// TIA Portal V15.1 export
// export: Created 2020-06-12T07:35:49.5849609Z, ExportSetting None, DisplayName Totally Integrated Automation Portal, DisplayVersion V15.1, DisplayName TIA Portal Openness, DisplayVersion V15.1, DisplayName STEP 7 Professional, DisplayVersion V15.1, DisplayName STEP 7 Safety, DisplayVersion V15.1, DisplayName WinCC Advanced, DisplayVersion V15.1
FUNCTION "MELT_Call" : Void   // FC91, FBD
{ S7_Optimized_Access := 'TRUE' }
// Melt control
// stored: SetENOAutomatically False
BEGIN

REGION Network 1: Melt time
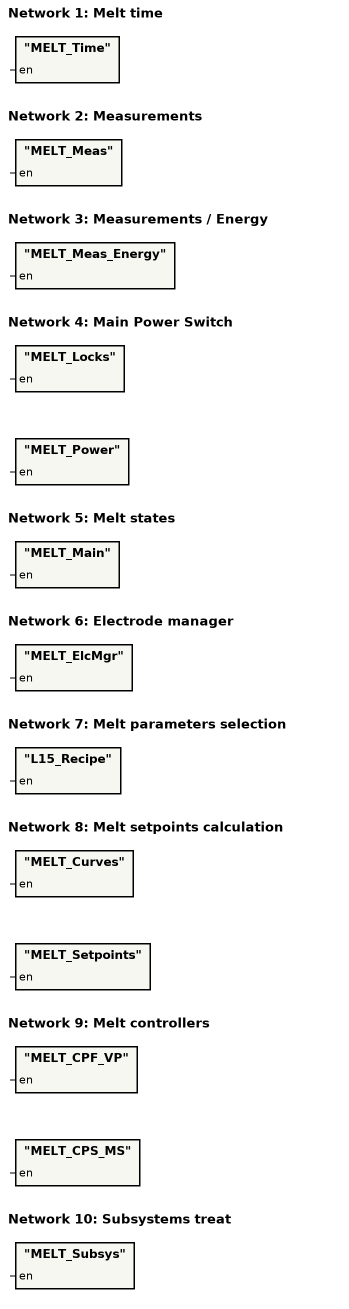
   "MELT_Time"();
END_REGION

REGION Network 2: Measurements
   "MELT_Meas"();
END_REGION

REGION Network 3: Measurements / Energy
   "MELT_Meas_Energy"();
END_REGION

REGION Network 4: Main Power Switch
   "MELT_Locks"();
   "MELT_Power"();
END_REGION

REGION Network 5: Melt states
   "MELT_Main"();
END_REGION

REGION Network 6: Electrode manager
   "MELT_ElcMgr"();
END_REGION

REGION Network 7: Melt parameters selection
   "L15_Recipe"();
END_REGION

REGION Network 8: Melt setpoints calculation
   "MELT_Curves"();
   "MELT_Setpoints"();
END_REGION

REGION Network 9: Melt controllers
   "MELT_CPF_VP"();
   "MELT_CPS_MS"();
END_REGION

REGION Network 10: Subsystems treat
   "MELT_Subsys"();
END_REGION

REGION Network 11: VISU Commands reset
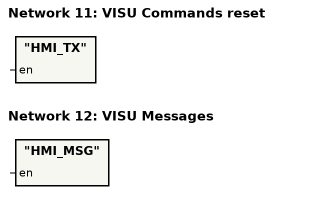
   "HMI_TX"();
END_REGION

REGION Network 12: VISU Messages
   "HMI_MSG"();
END_REGION
END_FUNCTION
